PROGRAM MAIN
VAR
 
END_VAR

END_PROGRAM

(* stored: Version 1.1.0.1
   POU MAIN: Id {2a241386-596a-4682-94af-4f5353c7e767}, SpecialFunc None *)
